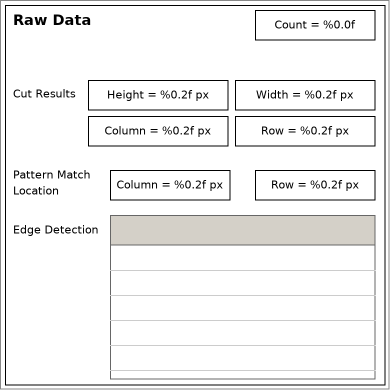
VISUALIZATION Manual_Camera_RawData  // 390x390
    Rectangle (5,5 380x380)
    Label (10,5 297x30), "Raw Data"
    Rectangle (255,10 120x30), "Count = %0.0f", text variable: MAIN.fbSlitter.Camera.CameraData.Results.Count
    Rectangle (110,170 120x30), "Column = %0.2f px", text variable: MAIN.fbSlitter.Camera.CameraData.Results.PatternMatchColumn
    Rectangle (255,170 120x30), "Row = %0.2f px", text variable: MAIN.fbSlitter.Camera.CameraData.Results.PatternMatchRow
    Rectangle (88,116 140x30), "Column = %0.2f px", text variable: MAIN.fbSlitter.Camera.CameraData.Results.LocationInX
    Rectangle (235,116 140x30), "Row = %0.2f px", text variable: MAIN.fbSlitter.Camera.CameraData.Results.LocationInY
    Rectangle (88,80 140x30), "Height = %0.2f px", text variable: MAIN.fbSlitter.Camera.CameraData.Results.HeightMeasurement
    Rectangle (235,80 140x30), "Width = %0.2f px", text variable: MAIN.fbSlitter.Camera.CameraData.Results.WidthMeasurement
    Label (10,215 101x30), "Edge Detection"
    Table (110,215 265x164), data array: MAIN.fbSlitter.Camera._displayVisionPts
        p1128707560: GVL.NumberVisionPoints
        p3854506369: MAIN.fbSlitter.Camera._displayVisionPts[1,INDEX]
        p1892666644: MAIN.fbSlitter.Camera._displayVisionPts[2,INDEX]
        p2232123230: Column
        p511219082: Row
    Group (10,160 96x46)
        Label (0,0 96x30), "Pattern Match"
        Label (0,16 96x30), "Location"
    Label (10,79 101x30), "Cut Results"
END_VISUALIZATION

(* stored: Version 1.1.0.1, ProductVersion 3.1.4024.3
   Visu Manual_Camera_RawData: Id {c6708db4-42a1-468f-b0fa-82a8f446d77b} *)
